(* IEC 61131-3 sources: AXOpen/src/components.rexroth.drives/app/src/Sandbox, 1 file *)

(* ---- SandboxContext.st ---- *)
USING AXOpen.Components.Rexroth.Drives;
USING System.Timer;

NAMESPACE AXOpen.Components.Rexroth.Drives
    {S7.extern=ReadWrite}
    CLASS SandboxContext EXTENDS AXOpen.Core.AxoContext
        VAR PUBLIC
            {#ix-attr:[Container(Layout.Wrap)]}
            {#ix-set:AttributeName = "<#Activate manual control#>"}
            _manualControl  : BOOL := TRUE;
            {#ix-set:AttributeName = "<#Enable drive signal#>"}
            Enable     : BOOL := TRUE;
            {#ix-set:AttributeName = "<#Enable in positive direction signal#>"}
            EnablePositive : BOOL := TRUE;
            {#ix-set:AttributeName = "<#Enable in positive negative signal#>"}
            EnableNegative   : BOOL := TRUE;
            {#ix-attr:[Container(Layout.Stack)]}
            IndraDrive  : AXOpen.Components.Rexroth.Drives.AxoIndraDrive;
            {#ix-attr:[Container(Layout.Stack)]}
            CtrlXdrive : AXOpen.Components.Rexroth.Drives.AxoCtrlxDriveXsc;
            _rootObject :   AxoObject;
        END_VAR

        VAR PUBLIC
            NumberOfCycles : ULINT := ULINT#10;
            Position1: LREAL := LREAL#10.0;
            Position2: LREAL := LREAL#15.0;
            Velocity : LREAL := LREAL#10.0;
            MaxTime : TIME := TIME#5m;
            Sequencer : AxoSequencer;
            Steps : ARRAY[0..15] OF AXOpen.Core.AxoStep;
            StartTime : LTIME;
            EndTime : LTIME;
            Cycle : ULINT;
            TotalDuration : LTIME;
            DurationPerCycle : LTIME;

            Timer : OnDelay;
            RunTimer : BOOL;
        END_VAR

        METHOD PROTECTED OVERRIDE Main
            RETURN;
            THIS.InitializeRootObject(_rootObject);
            IF(_manualControl) THEN
                IndraDrive.ActivateManualControl();
            END_IF;

            IndraDrive.Run(inParent               :=  _rootObject,
                            hwID                :=  HwIdentifiers#rexroth_indradrive_HwID,
                            Enable              :=  Enable,
                            EnablePositive      :=  EnablePositive,
                            EnableNegative      :=  EnableNegative);

            THIS.UseInSequencerIndraDrive();

            CtrlXdrive.Run(inParent               :=  _rootObject,
                            hwID                :=  HwIdentifiers#rexroth_ctrlx_drive_HwID,
                            Enable              :=  Enable,
                            EnablePositive      :=  EnablePositive,
                            EnableNegative      :=  EnableNegative);

            THIS.UseInSequencerCtrlXdrive();

        END_METHOD

        METHOD PRIVATE UseInSequencerIndraDrive

            Sequencer.Run(_rootObject);
            Sequencer.Open();
            Sequencer.SequenceMode := eAxoSequenceMode#RunOnce;

            Timer(signal := RunTimer, duration := MaxTime);

            IF(Steps[0].Execute(Sequencer, 'Restore')) THEN
                _manualControl := FALSE;
                Enable := FALSE;
                EnablePositive := FALSE;
                EnableNegative := FALSE;
                IndraDrive.Restore();
                Sequencer.MoveNext();
                RunTimer := FALSE;
                RETURN;
            END_IF;

            IF(Steps[1].Execute(Sequencer, 'Reset drive')) THEN
                RunTimer := TRUE;
                IF(IndraDrive.AxoReset().IsDone()) THEN
                    Sequencer.MoveNext();
                END_IF;
            END_IF;

            IF(Steps[2].Execute(Sequencer, 'Enable drive')) THEN
                Enable := TRUE;
                EnablePositive := TRUE;
                EnableNegative := TRUE;
                IF(IndraDrive.AxoPower_Status) THEN
                    Sequencer.MoveNext();
                END_IF;
            END_IF;

            IF(Steps[3].Execute(Sequencer, 'Drive homming')) THEN
                IF(IndraDrive.AxoHome(  Position        :=  LREAL#5.0,
                                            HommingMode     :=  INT#551,
                                            Velocity        :=  LREAL#1.0,
                                            Acceleration    :=  LREAL#50.0,
                                            Deceleration    :=  LREAL#50.0
                                            ).IsDone()) THEN
                    Sequencer.MoveNext();
                END_IF;
            END_IF;

            IF(Steps[4].Execute(Sequencer, 'Move absolute to start Position2')) THEN
                IF(IndraDrive.AxoMoveAbsolute(   Position        :=  Position2,
                                                    Velocity        :=  Velocity,
                                                    Acceleration    :=  LREAL#50.0,
                                                    Deceleration    :=  LREAL#50.0,
                                                    Jerk            :=  LREAL#150000.0
                                                    ).IsDone()) THEN
                    Sequencer.MoveNext();
                END_IF;
            END_IF;

            IF(Steps[5].Execute(Sequencer, 'Restore component to be able to trigger next move absolute in the same PLC cycle')) THEN
                IndraDrive.Restore();

                StartTime := Timer.elapsedTime;
                EndTime := StartTime;
                Cycle := ULINT#0;
                TotalDuration := LTIME#0s;
                DurationPerCycle := LTIME#0s;

                Sequencer.MoveNext();
            END_IF;

            IF(Steps[6].Execute(Sequencer, 'Move absolute to Position1')) THEN
                IF(IndraDrive.AxoMoveAbsolute(   Position        :=  Position1,
                                                    Velocity        :=  Velocity,
                                                    Acceleration    :=  LREAL#50.0,
                                                    Deceleration    :=  LREAL#50.0,
                                                    Jerk            :=  LREAL#150000.0
                                                    ).IsDone()) THEN
                    Sequencer.MoveNext();
                END_IF;
            END_IF;

            IF(Steps[7].Execute(Sequencer, 'Restore component to be able to trigger next move absolute in the same PLC cycle')) THEN
                IndraDrive.Restore();
                Sequencer.MoveNext();
            END_IF;

            IF(Steps[8].Execute(Sequencer, 'Move absolute to Position2')) THEN
                IF(IndraDrive.AxoMoveAbsolute(   Position        :=  Position2,
                                                    Velocity        :=  Velocity,
                                                    Acceleration    :=  LREAL#50.0,
                                                    Deceleration    :=  LREAL#50.0,
                                                    Jerk            :=  LREAL#150000.0
                                                    ).IsDone()) THEN
                    Sequencer.MoveNext();
                END_IF;
            END_IF;

            IF(Steps[9].Execute(Sequencer, 'Restore component to be able to trigger next move absolute in the same PLC cycle')) THEN
                IndraDrive.Restore();
                Sequencer.MoveNext();
            END_IF;

            IF(Steps[10].Execute(Sequencer, 'Repetition')) THEN
                Cycle := Cycle + ULINT#1;
                EndTime :=  Timer.elapsedTime;
                TotalDuration := EndTime - StartTime;
                DurationPerCycle := TotalDuration / Cycle;
                IF(Cycle >= NumberOfCycles) THEN
                    Sequencer.MoveNext();
                ELSE
                    Sequencer.RequestStep(Steps[6]);
                END_IF;
            END_IF;

            IF(Steps[11].Execute(Sequencer, 'Disable drive')) THEN
                Enable := FALSE;
                EnablePositive := FALSE;
                EnableNegative := FALSE;
                IF(NOT IndraDrive.AxoPower_Status) THEN
                    Sequencer.CompleteSequence();
                END_IF;
            END_IF;

            IF(Steps[12].Execute(Sequencer, 'Reset drive')) THEN
                IF(IndraDrive.AxoReset().IsDone()) THEN
                    Sequencer.MoveNext();
                END_IF;
            END_IF;

            IF(Steps[13].Execute(Sequencer, 'Restore')) THEN
                IndraDrive.Restore();
                Sequencer.CompleteSequence();
            END_IF;
        END_METHOD
        METHOD PRIVATE UseInSequencerCtrlXdrive

            Sequencer.Run(_rootObject);
            Sequencer.Open();
            Sequencer.SequenceMode := eAxoSequenceMode#RunOnce;

            Timer(signal := RunTimer, duration := MaxTime);

            IF(Steps[0].Execute(Sequencer, 'Restore')) THEN
                _manualControl := FALSE;
                Enable := FALSE;
                EnablePositive := FALSE;
                EnableNegative := FALSE;
                CtrlXdrive.Restore();
                Sequencer.MoveNext();
                RunTimer := FALSE;
                RETURN;
            END_IF;

            IF(Steps[1].Execute(Sequencer, 'Reset drive')) THEN
                RunTimer := TRUE;
                IF(CtrlXdrive.AxoReset().IsDone()) THEN
                    Sequencer.MoveNext();
                END_IF;
            END_IF;

            IF(Steps[2].Execute(Sequencer, 'Enable drive')) THEN
                Enable := TRUE;
                EnablePositive := TRUE;
                EnableNegative := TRUE;
                IF(CtrlXdrive.AxoPower_Status) THEN
                    Sequencer.MoveNext();
                END_IF;
            END_IF;

            IF(Steps[3].Execute(Sequencer, 'Drive homming')) THEN
                IF(CtrlXdrive.AxoHome(  Position        :=  LREAL#5.0,
                                            HommingMode     :=  INT#551,
                                            Velocity        :=  LREAL#1.0,
                                            Acceleration    :=  LREAL#50.0,
                                            Deceleration    :=  LREAL#50.0
                                            ).IsDone()) THEN
                    Sequencer.MoveNext();
                END_IF;
            END_IF;

            IF(Steps[4].Execute(Sequencer, 'Move absolute to start Position2')) THEN
                IF(CtrlXdrive.AxoMoveAbsolute(   Position        :=  Position2,
                                                    Velocity        :=  Velocity,
                                                    Acceleration    :=  LREAL#50.0,
                                                    Deceleration    :=  LREAL#50.0,
                                                    Jerk            :=  LREAL#150000.0
                                                    ).IsDone()) THEN
                    Sequencer.MoveNext();
                END_IF;
            END_IF;

            IF(Steps[5].Execute(Sequencer, 'Restore component to be able to trigger next move absolute in the same PLC cycle')) THEN
                CtrlXdrive.Restore();

                StartTime := Timer.elapsedTime;
                EndTime := StartTime;
                Cycle := ULINT#0;
                TotalDuration := LTIME#0s;
                DurationPerCycle := LTIME#0s;

                Sequencer.MoveNext();
            END_IF;

            IF(Steps[6].Execute(Sequencer, 'Move absolute to Position1')) THEN
                IF(CtrlXdrive.AxoMoveAbsolute(   Position        :=  Position1,
                                                    Velocity        :=  Velocity,
                                                    Acceleration    :=  LREAL#50.0,
                                                    Deceleration    :=  LREAL#50.0,
                                                    Jerk            :=  LREAL#150000.0
                                                    ).IsDone()) THEN
                    Sequencer.MoveNext();
                END_IF;
            END_IF;

            IF(Steps[7].Execute(Sequencer, 'Restore component to be able to trigger next move absolute in the same PLC cycle')) THEN
                CtrlXdrive.Restore();
                Sequencer.MoveNext();
            END_IF;

            IF(Steps[8].Execute(Sequencer, 'Move absolute to Position2')) THEN
                IF(CtrlXdrive.AxoMoveAbsolute(   Position        :=  Position2,
                                                    Velocity        :=  Velocity,
                                                    Acceleration    :=  LREAL#50.0,
                                                    Deceleration    :=  LREAL#50.0,
                                                    Jerk            :=  LREAL#150000.0
                                                    ).IsDone()) THEN
                    Sequencer.MoveNext();
                END_IF;
            END_IF;

            IF(Steps[9].Execute(Sequencer, 'Restore component to be able to trigger next move absolute in the same PLC cycle')) THEN
                CtrlXdrive.Restore();
                Sequencer.MoveNext();
            END_IF;

            IF(Steps[10].Execute(Sequencer, 'Repetition')) THEN
                Cycle := Cycle + ULINT#1;
                EndTime :=  Timer.elapsedTime;
                TotalDuration := EndTime - StartTime;
                DurationPerCycle := TotalDuration / Cycle;
                IF(Cycle >= NumberOfCycles) THEN
                    Sequencer.MoveNext();
                ELSE
                    Sequencer.RequestStep(Steps[6]);
                END_IF;
            END_IF;

            IF(Steps[11].Execute(Sequencer, 'Disable drive')) THEN
                Enable := FALSE;
                EnablePositive := FALSE;
                EnableNegative := FALSE;
                IF(NOT CtrlXdrive.AxoPower_Status) THEN
                    Sequencer.CompleteSequence();
                END_IF;
            END_IF;

            IF(Steps[12].Execute(Sequencer, 'Reset drive')) THEN
                IF(CtrlXdrive.AxoReset().IsDone()) THEN
                    Sequencer.MoveNext();
                END_IF;
            END_IF;

            IF(Steps[13].Execute(Sequencer, 'Restore')) THEN
                CtrlXdrive.Restore();
                Sequencer.CompleteSequence();
            END_IF;
        END_METHOD
    END_CLASS
END_NAMESPACE
